FUNCTION_BLOCK Valve EXTENDS BaseValve
VAR_INPUT
	IO_Open: REFERENCE TO DigitalOutput;
	IO_FB1, IO_FB2: REFERENCE TO DigitalInput;
END_VAR
VAR_OUTPUT
END_VAR
VAR
	ValveMonitor: ValveMonitor; 
	Error: BOOL;
END_VAR

ValveMonitor(Valve := Open, FB1 := IsOpen, FB2 := IsClosed);
Error := ValveMonitor.Error;

END_FUNCTION_BLOCK

(* stored: Version 1.1.0.1, ProductVersion 3.1.4024.3
   POU Valve: Id {f79b007e-61a9-4d86-9184-28e3572ebdbb}, SpecialFunc None *)
